FUNCTION_BLOCK ParallelUnits
VAR_INPUT
	EN: BOOL;
	Tags: REFERENCE TO AdsTagsParallelUnits;
	Parameters: REFERENCE TO GreenMasterBaseParameters;
END_VAR
VAR_OUTPUT
END_VAR
VAR
	LocalAmsNumber: LINT;
	RemoteAmsNumber: LINT;
	RemoteOrderToSend: RemoteOrder;
	RemoteStatusData: RemoteStatusData;
	Week: WORD;
	FirstTime: BOOL;
	HostName: FB_GetHostName;
	FoundHost: BOOL;
	StateTime: Timer;
	RemoteActive: BOOL;
	InstantaneousDualNeeded: BOOL;
	DualNeeded: BOOL;
	DualNeededTON: TON;
	DualNeededTOF: TOF;
	Runnable: BOOL;
	RemoteValidTOF: TOF;
	AddWeekTest: WORD;
	TransferOk: BOOL;
	TransferTON: TON;
	TempSP: LREAL;
	SupplyAirSetPointAdjustmentFB: SetPointAdjustmentFB;
	ExtractAirSetPointAdjustmentFB: SetPointAdjustmentFB;
	SupplyAirSetPointAdjustmentFB_HighSpeed: SetPointAdjustmentFB;
	ExtractAirSetPointAdjustmentFB_HighSpeed: SetPointAdjustmentFB;
	StandaloneSupplyAirSetPointAdjustmentFB: SetPointAdjustmentFB;
	StandaloneExtractAirSetPointAdjustmentFB: SetPointAdjustmentFB;
	StandaloneSupplyAirSetPointAdjustmentFB_HighSpeed: SetPointAdjustmentFB;
	StandaloneExtractAirSetPointAdjustmentFB_HighSpeed: SetPointAdjustmentFB;
END_VAR

IF NOT FirstTime THEN
	HostName(bExecute := TRUE);
	IF NOT HostName.bBusy THEN	
		FoundHost := FALSE;
		// E6
		IF F_ToUCase(HostName.sHostName) = 'STU_E6-LB01' THEN
			Tags.Settings.RemoteAmsId := '10.138.21.151.1.1';
			Tags.Status.isMaster := TRUE;
			FoundHost := TRUE;
		ELSIF F_ToUCase(HostName.sHostName) = 'STU_E6-LB02' THEN
			Tags.Settings.RemoteAmsId := '10.138.21.150.1.1';
			Tags.Status.isMaster := FALSE;
			FoundHost := TRUE;
		END_IF
		// E1
		IF F_ToUCase(HostName.sHostName) = 'STU_E1-LB01' THEN
			Tags.Settings.RemoteAmsId := '10.138.21.153.1.1';
			Tags.Status.isMaster := TRUE;
			FoundHost := TRUE;
		ELSIF F_ToUCase(HostName.sHostName) = 'STU_E1-LB02' THEN
			Tags.Settings.RemoteAmsId := '10.138.21.152.1.1';
			Tags.Status.isMaster := FALSE;
			FoundHost := TRUE;
		END_IF
		// DIGINET Test system
		IF F_ToUCase(HostName.sHostName) = 'DIGINET-1' THEN
			Tags.Settings.RemoteAmsId := '5.102.41.153.1.1';
			Tags.Status.isMaster := TRUE;
			FoundHost := TRUE;
		ELSIF F_ToUCase(HostName.sHostName) = 'DIGINET-2' THEN
			Tags.Settings.RemoteAmsId := '5.73.47.143.1.1';
			Tags.Status.isMaster := FALSE;
			FoundHost := TRUE;
		END_IF
		// NIBE AirSite Test system
		IF F_ToUCase(HostName.sHostName) = 'AIRPLC-DEMO' THEN
			Tags.Settings.RemoteAmsId := '5.102.42.161.1.1';
			Tags.Status.isMaster := TRUE;
			FoundHost := TRUE;
		ELSIF F_ToUCase(HostName.sHostName) = 'CX-662AA1' THEN
			Tags.Settings.RemoteAmsId := '10.133.0.22.1.1';
			Tags.Status.isMaster := FALSE;
			FoundHost := TRUE;
		END_IF
		IF NOT FoundHost THEN
			Tags.Status.isMaster := TRUE;			
		END_IF
		Tags.Status.isSlave := NOT Tags.Status.isMaster;
		// First time or remote AMS ID changed
		FirstTime := TRUE;
	END_IF
END_IF
StateTime();
Runnable := Parameters.System.Operation.State = SystemStates.Run;
IF Runnable THEN
	IF NOT InstantaneousDualNeeded THEN
		IF (Parameters.Regulation.SupplyAir.Control.CV > Tags.Settings.StandaloneMaxFan) OR
			(Parameters.Regulation.ExtractAir.Control.CV > Tags.Settings.StandaloneMaxFan) OR
			(RemoteStatusData.RemoteStatus.SupplyFanSpeed > Tags.Settings.StandaloneMaxFan) OR
			(RemoteStatusData.RemoteStatus.ExtractFanSpeed > Tags.Settings.StandaloneMaxFan) THEN
			InstantaneousDualNeeded := TRUE;
		END_IF
	ELSE
		IF (Parameters.Regulation.SupplyAir.Control.CV < Tags.Settings.DualMinFan) AND
			(Parameters.Regulation.ExtractAir.Control.CV < Tags.Settings.DualMinFan) AND
			(RemoteStatusData.RemoteStatus.SupplyFanSpeed < Tags.Settings.DualMinFan) AND
			(RemoteStatusData.RemoteStatus.ExtractFanSpeed < Tags.Settings.DualMinFan) THEN
			InstantaneousDualNeeded := FALSE;
		END_IF
	END_IF
	DualNeededTON(IN := InstantaneousDualNeeded, PT := T#5M);
	DualNeededTOF(IN := InstantaneousDualNeeded, PT := T#5M);
	IF NOT DualNeeded THEN
		IF DualNeededTON.Q THEN
			DualNeeded := TRUE;
		END_IF
	ELSE
		IF NOT DualNeededTOF.Q THEN
			DualNeeded := FALSE;
		END_IF
	END_IF
END_IF
Week := F_GetWeekOfTheYear(NowDT()) + AddWeekTest;;
RemoteValidTOF(IN := RemoteStatusData.Valid, PT := T#10S); 
RemoteActive := RemoteValidTOF.Q AND RemoteStatusData.RemoteStatus.IsRunning;
Tags.Status.SupplyFanSpeed := Parameters.Regulation.SupplyAir.Control.CV;
Tags.Status.ExtractFanSpeed := Parameters.Regulation.ExtractAir.Control.CV;
Tags.Status.IsRunning := Parameters.System.Operation.State = SystemStates.Run;
Tags.Status.ResetAlarm := Parameters.IO.DIn.ResetAlarm;
Tags.Status.Fire := Main.GreenMaster.FireAlarm();
Tags.Status.Freeze := Parameters.Alarm.Active.A.Freeze;
IF RemoteActive THEN
	Tags.Status.PressureSupplyCSP := GetSetPointSupply();
	Tags.Status.PressureExtractCSP := GetSetPointExtract();
ELSE
	Tags.Status.PressureSupplyCSP := GetStandaloneSetPointSupply();
	Tags.Status.PressureExtractCSP := GetStandaloneSetPointExtract();
END_IF

IF FirstTime THEN
	MasterSlave();
END_IF
IF EN THEN
	TransferTON(IN := TRUE, PT := T#1S);
	IF TransferTON.Q THEN
		TransferTON(IN := FALSE);
		RemoteStatusData := ReadFromRemote();
		IF RemoteStatusData.Valid THEN
			IF RemoteStatusData.RemoteStatus.ResetAlarm THEN
				Parameters.Alarm.Control.ResetAlarms := TRUE;
			END_IF
			RemoteOrderToSend.Counter := RemoteOrderToSend.Counter + 1;
			IF Tags.Status.IsMaster THEN
				RemoteOrderToSend.TimeChannels := Parameters.System.Operation.TimeChannels;
				RemoteOrderToSend.TemperatureControl := Parameters.Regulation.Temperature.Control;		
				RemoteOrderToSend.SupplyAirControl := Parameters.Regulation.SupplyAir.Control;		
				RemoteOrderToSend.ExtractAirControl := Parameters.Regulation.ExtractAir.Control;
				RemoteOrderToSend.TemperatureSetPointAdjustment := Parameters.Regulation.Temperature.SetPointAdjustment;
				RemoteOrderToSend.SupplyAirSetPointAdjustment := Parameters.Regulation.SupplyAir.SetPointAdjustment;
				RemoteOrderToSend.ExtractAirSetPointAdjustment := Parameters.Regulation.ExtractAir.SetPointAdjustment;
				RemoteOrderToSend.NightCoolingRequest := Parameters.Regulation.NightCoolingRequest;
			END_IF
			TransferOk := TransferToRemote(sNetId := Tags.Settings.RemoteAmsId, Src := RemoteOrderToSend, Dest := 'ADS_ParallelUnits.Tags.Settings.RemoteOrder');	
			IF TransferOk AND Tags.Status.IsSlave THEN
				Parameters.System.Operation.TimeChannels := Tags.Settings.RemoteOrder.TimeChannels;		
				Parameters.Regulation.Temperature.Control.SP := Tags.Settings.RemoteOrder.TemperatureControl.SP;		
				Parameters.Regulation.Temperature.Control.SP_HighSpeed := Tags.Settings.RemoteOrder.TemperatureControl.SP_HighSpeed;		
				Parameters.Regulation.SupplyAir.Control.SP := Tags.Settings.RemoteOrder.SupplyAirControl.SP;		
				Parameters.Regulation.SupplyAir.Control.SP_HighSpeed := Tags.Settings.RemoteOrder.SupplyAirControl.SP_HighSpeed;		
				Parameters.Regulation.ExtractAir.Control.SP := Tags.Settings.RemoteOrder.ExtractAirControl.SP;		
				Parameters.Regulation.ExtractAir.Control.SP_HighSpeed := Tags.Settings.RemoteOrder.ExtractAirControl.SP_HighSpeed;		
				Parameters.Regulation.Temperature.SetPointAdjustment := Tags.Settings.RemoteOrder.TemperatureSetPointAdjustment;		
				Parameters.Regulation.SupplyAir.SetPointAdjustment := Tags.Settings.RemoteOrder.SupplyAirSetPointAdjustment;		
				Parameters.Regulation.ExtractAir.SetPointAdjustment := Tags.Settings.RemoteOrder.ExtractAirSetPointAdjustment;	
				Parameters.Regulation.NightCoolingRequest := Tags.Settings.RemoteOrder.NightCoolingRequest;
			END_IF
		ELSE
			IF Tags.Status.IsSlave THEN
				Parameters.Regulation.NightCoolingRequest := FALSE;
			END_IF
		END_IF		
	END_IF
END_IF

METHOD GetAmsNumbers : BOOL
VAR_INPUT
END_VAR
VAR_INST
	LocalAddrBytes: AMSNETID;
	RemoteAddrBytes: AMSNETID;	
	FB_GetLocalAmsNetId: FB_GetLocalAmsNetId;
	UsedRemoteAmsId: string := '???';
END_VAR
IF Tags.Settings.RemoteAmsId <> UsedRemoteAmsId THEN
	UsedRemoteAmsId := Tags.Settings.RemoteAmsId;
	RemoteAddrBytes := F_ScanAmsNetIds(Tags.Settings.RemoteAmsId);
	FB_GetLocalAmsNetId(bExecute := TRUE, AddrBytes => LocalAddrBytes);
	FB_GetLocalAmsNetId(bExecute := FALSE);
	IF NOT FB_GetLocalAmsNetId.bBusy AND NOT FB_GetLocalAmsNetId.bError THEN			
		LocalAmsNumber := 	
						SHL(TO_LINT(LocalAddrBytes[0]),  40) + 
						SHL(TO_LINT(LocalAddrBytes[1]),  32) + 
						SHL(TO_LINT(LocalAddrBytes[2]),  24) + 
						SHL(TO_LINT(LocalAddrBytes[3]), 16) + 
						SHL(TO_LINT(LocalAddrBytes[4]), 8) + 
						TO_LINT(LocalAddrBytes[5]); 
		RemoteAmsNumber := 	
						SHL(TO_LINT(RemoteAddrBytes[0]),  40) + 
						SHL(TO_LINT(RemoteAddrBytes[1]),  32) + 
						SHL(TO_LINT(RemoteAddrBytes[2]),  24) + 
						SHL(TO_LINT(RemoteAddrBytes[3]), 16) + 
						SHL(TO_LINT(RemoteAddrBytes[4]), 8) + 
						TO_LINT(RemoteAddrBytes[5]); 
	END_IF
	GetAmsNumbers := TRUE;
ELSE 
	GetAmsNumbers := FALSE;
END_IF
END_METHOD

METHOD GetSetPointExtract : REAL
VAR_INPUT
END_VAR
VAR
	TempSP: REAL;
END_VAR
IF Parameters.Regulation.NightCooling OR Parameters.IO.DIn.ExtendedOperation OR Parameters.System.Operation.TimeChannels.HighSpeed THEN
	TempSP := Tags.Settings.PressureExtractSP_HighSpeed;
	ExtractAirSetPointAdjustmentFB_HighSpeed(X := Parameters.Regulation.CompensationTemperature, SetPointAdjustment := Tags.Settings.ExtractAirSetPointAdjustment_HighSpeed);
	GetSetPointExtract := TO_REAL(Tags.Settings.ExtractAirSetPointAdjustment_HighSpeed.Y) + TempSP;
ELSE
	TempSP := Tags.Settings.PressureExtractSP;
	ExtractAirSetPointAdjustmentFB(X := Parameters.Regulation.CompensationTemperature, SetPointAdjustment := Tags.Settings.ExtractAirSetPointAdjustment);
	GetSetPointExtract := TO_REAL(Tags.Settings.ExtractAirSetPointAdjustment.Y) + TempSP;
END_IF
END_METHOD

METHOD GetSetPointSupply : REAL
VAR_INPUT
END_VAR
VAR
	TempSP: REAL;
END_VAR
IF Parameters.Regulation.NightCooling OR Parameters.IO.DIn.ExtendedOperation OR Parameters.System.Operation.TimeChannels.HighSpeed THEN
	TempSP := Tags.Settings.PressureSupplySP_HighSpeed;
	SupplyAirSetPointAdjustmentFB_HighSpeed(X := Parameters.Regulation.CompensationTemperature, SetPointAdjustment := Tags.Settings.SupplyAirSetPointAdjustment_HighSpeed);
	GetSetPointSupply := TO_REAL(Tags.Settings.SupplyAirSetPointAdjustment_HighSpeed.Y) + TempSP;
ELSE
	TempSP := Tags.Settings.PressureSupplySP;
	SupplyAirSetPointAdjustmentFB(X := Parameters.Regulation.CompensationTemperature, SetPointAdjustment := Tags.Settings.SupplyAirSetPointAdjustment);
	GetSetPointSupply := TO_REAL(Tags.Settings.SupplyAirSetPointAdjustment.Y) + TempSP;
END_IF
END_METHOD

METHOD GetStandaloneSetPointExtract : REAL
VAR_INPUT
END_VAR
VAR
	TempSP: REAL;
END_VAR
IF Parameters.Regulation.NightCooling OR Parameters.IO.DIn.ExtendedOperation OR Parameters.System.Operation.TimeChannels.HighSpeed THEN
	TempSP := Tags.Settings.StandalonePressureExtractSP_HighSpeed;
	StandaloneExtractAirSetPointAdjustmentFB_HighSpeed(X := Parameters.Regulation.CompensationTemperature, SetPointAdjustment := Tags.Settings.StandaloneExtractAirSetPointAdjustment_HighSpeed);
	GetStandaloneSetPointExtract := TO_REAL(Tags.Settings.StandaloneExtractAirSetPointAdjustment_HighSpeed.Y) + TempSP;
ELSE
	TempSP := Tags.Settings.StandalonePressureExtractSP;
	StandaloneExtractAirSetPointAdjustmentFB(X := Parameters.Regulation.CompensationTemperature, SetPointAdjustment := Tags.Settings.StandaloneExtractAirSetPointAdjustment);
	GetStandaloneSetPointExtract := TO_REAL(Tags.Settings.StandaloneExtractAirSetPointAdjustment.Y) + TempSP;
END_IF
END_METHOD

METHOD GetStandaloneSetPointSupply : REAL
VAR_INPUT
END_VAR
VAR
	TempSP: REAL;
END_VAR
IF Parameters.Regulation.NightCooling OR Parameters.IO.DIn.ExtendedOperation OR Parameters.System.Operation.TimeChannels.HighSpeed THEN
	TempSP := Tags.Settings.StandalonePressureSupplySP_HighSpeed;
	StandaloneSupplyAirSetPointAdjustmentFB_HighSpeed(X := Parameters.Regulation.CompensationTemperature, SetPointAdjustment := Tags.Settings.StandaloneSupplyAirSetPointAdjustment_HighSpeed);
	GetStandaloneSetPointSupply := TO_REAL(Tags.Settings.StandaloneSupplyAirSetPointAdjustment_HighSpeed.Y) + TempSP;
ELSE
	TempSP := Tags.Settings.StandalonePressureSupplySP;
	StandaloneSupplyAirSetPointAdjustmentFB(X := Parameters.Regulation.CompensationTemperature, SetPointAdjustment := Tags.Settings.StandaloneSupplyAirSetPointAdjustment);
	GetStandaloneSetPointSupply := TO_REAL(Tags.Settings.StandaloneSupplyAirSetPointAdjustment.Y) + TempSP;
END_IF
END_METHOD

METHOD MasterSlave : BOOL
VAR_INPUT
END_VAR
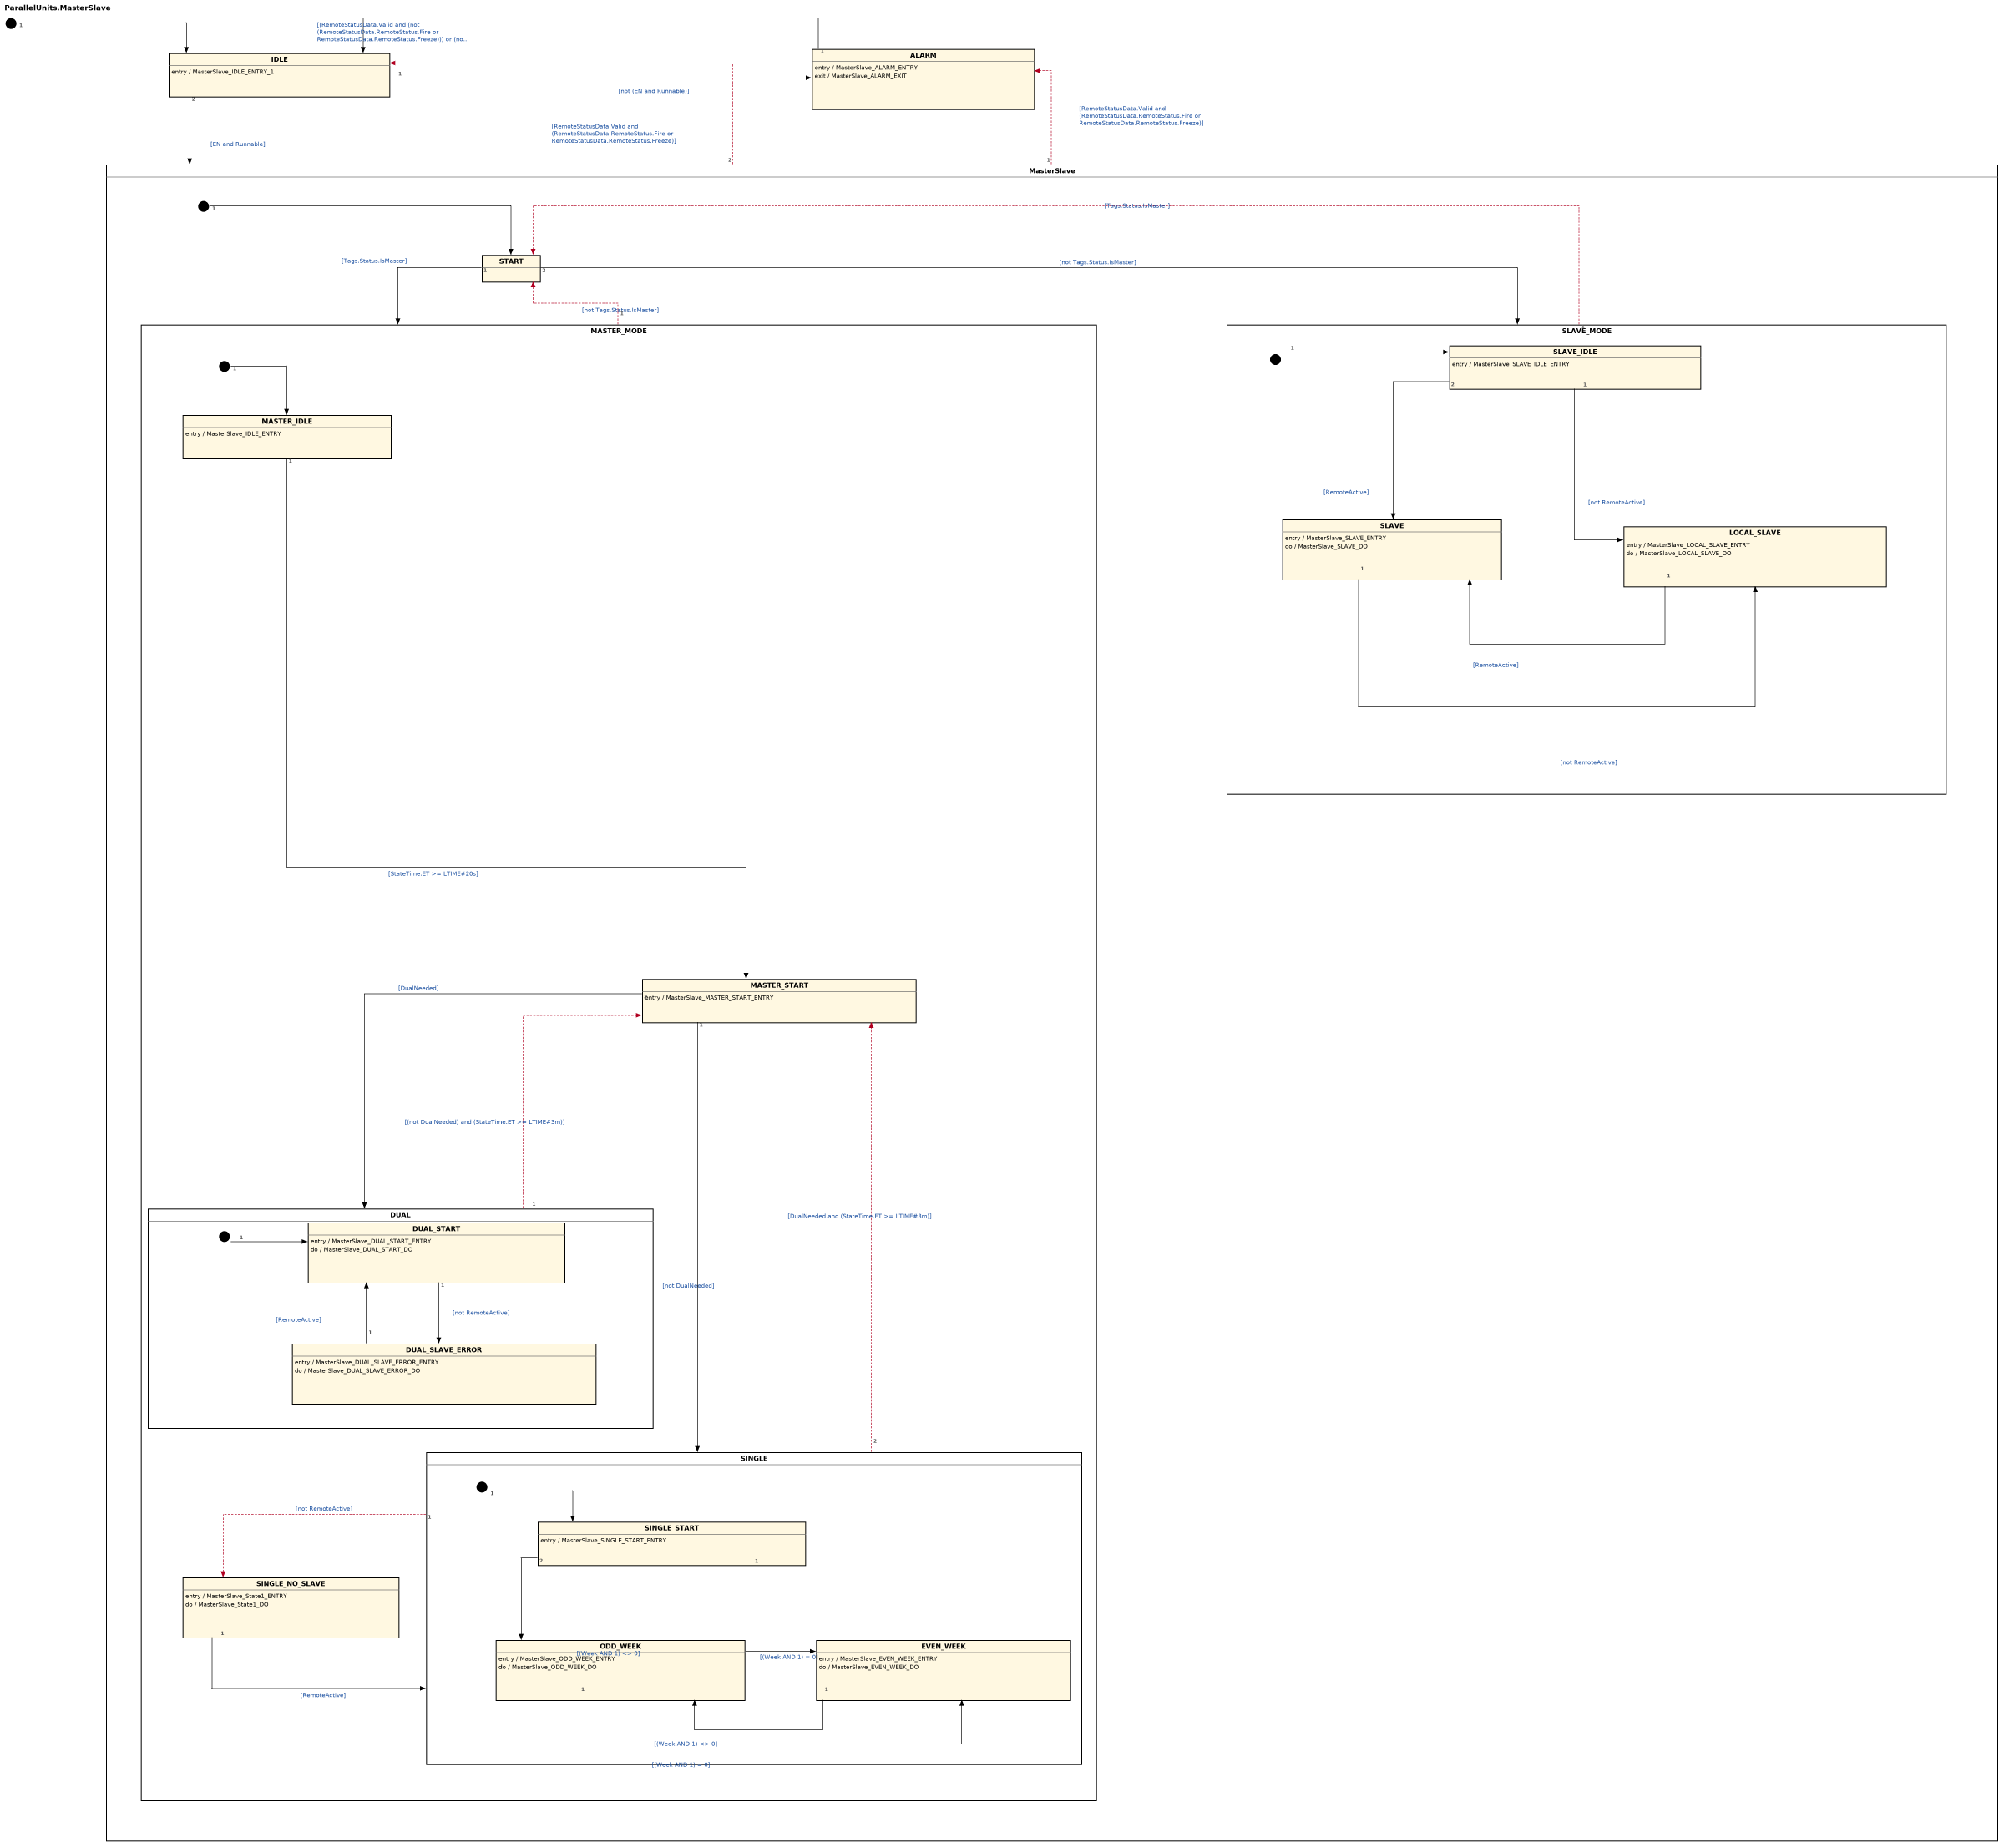
STATECHART MasterSlave  // abortable
    START StartState2
    STATE ALARM
        entry / MasterSlave_ALARM_ENTRY
        exit / MasterSlave_ALARM_EXIT
    STATE IDLE
        entry / MasterSlave_IDLE_ENTRY_1
    COMPOSITE STATE MasterSlave
        START StartState1
        STATE START
        COMPOSITE STATE MASTER_MODE
            START StartState6
            STATE MASTER_IDLE
                entry / MasterSlave_IDLE_ENTRY
            STATE MASTER_START
                entry / MasterSlave_MASTER_START_ENTRY
            COMPOSITE STATE DUAL
                START StartState4
                STATE DUAL_START
                    entry / MasterSlave_DUAL_START_ENTRY
                    do / MasterSlave_DUAL_START_DO
                STATE DUAL_SLAVE_ERROR
                    entry / MasterSlave_DUAL_SLAVE_ERROR_ENTRY
                    do / MasterSlave_DUAL_SLAVE_ERROR_DO
                StartState4 -> DUAL_START  // priority 1, on completion
                DUAL_START -> DUAL_SLAVE_ERROR [not RemoteActive] // priority 1
                DUAL_SLAVE_ERROR -> DUAL_START [RemoteActive] // priority 1
            END_STATE
            COMPOSITE STATE SINGLE
                START StartState3
                STATE SINGLE_START
                    entry / MasterSlave_SINGLE_START_ENTRY
                STATE ODD_WEEK
                    entry / MasterSlave_ODD_WEEK_ENTRY
                    do / MasterSlave_ODD_WEEK_DO
                STATE EVEN_WEEK
                    entry / MasterSlave_EVEN_WEEK_ENTRY
                    do / MasterSlave_EVEN_WEEK_DO
                StartState3 -> SINGLE_START  // priority 1, on completion
                SINGLE_START -> EVEN_WEEK [(Week AND 1) = 0] // priority 1
                SINGLE_START -> ODD_WEEK [(Week AND 1) <> 0] // priority 2
                ODD_WEEK -> EVEN_WEEK [(Week AND 1) = 0] // priority 1
                EVEN_WEEK -> ODD_WEEK [(Week AND 1) <> 0] // priority 1
            END_STATE
            STATE SINGLE_NO_SLAVE
                entry / MasterSlave_State1_ENTRY
                do / MasterSlave_State1_DO
            StartState6 -> MASTER_IDLE  // priority 1, on completion
            MASTER_IDLE -> MASTER_START [StateTime.ET >= LTIME#20s] // priority 1
            MASTER_START -> SINGLE [not DualNeeded] // priority 1
            MASTER_START -> DUAL [DualNeeded] // priority 2
            DUAL -> MASTER_START [(not DualNeeded) and (StateTime.ET >= LTIME#3m)] // priority 1, exception
            SINGLE -> SINGLE_NO_SLAVE [not RemoteActive] // priority 1, exception
            SINGLE -> MASTER_START [DualNeeded and (StateTime.ET >= LTIME#3m)] // priority 2, exception
            SINGLE_NO_SLAVE -> SINGLE [RemoteActive] // priority 1
        END_STATE
        COMPOSITE STATE SLAVE_MODE
            START StartState5
            STATE SLAVE_IDLE
                entry / MasterSlave_SLAVE_IDLE_ENTRY
            STATE SLAVE
                entry / MasterSlave_SLAVE_ENTRY
                do / MasterSlave_SLAVE_DO
            STATE LOCAL_SLAVE
                entry / MasterSlave_LOCAL_SLAVE_ENTRY
                do / MasterSlave_LOCAL_SLAVE_DO
            StartState5 -> SLAVE_IDLE  // priority 1, on completion
            SLAVE_IDLE -> LOCAL_SLAVE [not RemoteActive] // priority 1
            SLAVE_IDLE -> SLAVE [RemoteActive] // priority 2
            SLAVE -> LOCAL_SLAVE [not RemoteActive] // priority 1
            LOCAL_SLAVE -> SLAVE [RemoteActive] // priority 1
        END_STATE
        StartState1 -> START  // priority 1, on completion
        START -> MASTER_MODE [Tags.Status.IsMaster] // priority 1
        START -> SLAVE_MODE [not Tags.Status.IsMaster] // priority 2
        MASTER_MODE -> START [not Tags.Status.IsMaster] // priority 1, exception
        SLAVE_MODE -> START [Tags.Status.IsMaster] // priority 1, exception
    END_STATE
    StartState2 -> IDLE  // priority 1, on completion
    ALARM -> IDLE [(RemoteStatusData.Valid and (not (RemoteStatusData.RemoteStatus.Fire or RemoteStatusData.RemoteStatus.Freeze))) or (not RemoteStatusData.Valid)] // priority 1
    IDLE -> ALARM [RemoteStatusData.Valid and (RemoteStatusData.RemoteStatus.Fire or RemoteStatusData.RemoteStatus.Freeze)] // priority 1
    IDLE -> MasterSlave [EN and Runnable] // priority 2
    MasterSlave -> ALARM [RemoteStatusData.Valid and (RemoteStatusData.RemoteStatus.Fire or RemoteStatusData.RemoteStatus.Freeze)] // priority 1, exception
    MasterSlave -> IDLE [not (EN and Runnable)] // priority 2, exception
END_STATECHART
END_METHOD

METHOD MasterSlave_ALARM_ENTRY : BOOL
VAR_INPUT
END_VAR
Parameters.System.Operation.EN := FALSE;
END_METHOD

METHOD MasterSlave_ALARM_EXIT : BOOL
VAR_INPUT
END_VAR
Parameters.System.Operation.EN := TRUE;
END_METHOD

METHOD MasterSlave_DUAL_SLAVE_ERROR_DO : BOOL
VAR_INPUT
END_VAR
Parameters.Regulation.SupplyAir.Control.SP := GetStandaloneSetPointSupply();
Parameters.Regulation.ExtractAir.Control.SP := GetStandaloneSetPointExtract();
END_METHOD

METHOD MasterSlave_DUAL_SLAVE_ERROR_ENTRY : BOOL
VAR_INPUT
END_VAR
Parameters.Regulation.SupplyAir.ControlMode := FanControlTypes.Pressure;
Parameters.Regulation.ExtractAir.ControlMode := FanControlTypes.Pressure;
END_METHOD

METHOD MasterSlave_DUAL_START_DO : BOOL
VAR_INPUT
END_VAR
Parameters.Regulation.SupplyAir.Control.SP := PidControlSupplyAir(Sync := FALSE, SyncCV := 0);
Parameters.Regulation.ExtractAir.Control.SP := PidControlExtractAir(Sync := FALSE, SyncCV := 0);
RemoteOrderToSend.SupplySP := Parameters.Regulation.SupplyAir.Control.SP;
RemoteOrderToSend.ExtractSP := Parameters.Regulation.ExtractAir.Control.SP;
END_METHOD

METHOD MasterSlave_DUAL_START_ENTRY : BOOL
VAR_INPUT
END_VAR
StateTime.Restart();
Parameters.IO.DOut.T_QM2 := TRUE;
Parameters.IO.DOut.F_QM1 := TRUE;	
Parameters.Regulation.SupplyAir.ControlMode := FanControlTypes.Const;
Parameters.Regulation.ExtractAir.ControlMode := FanControlTypes.Const;
PidControlSupplyAir(Sync := FALSE, SyncCV := 0.55);
PidControlExtractAir(Sync := FALSE, SyncCV := 0.65);
PidControlSupplyAir(Sync := TRUE, SyncCV := 0.55);
PidControlExtractAir(Sync := TRUE, SyncCV := 0.65);
END_METHOD

METHOD MasterSlave_EVEN_WEEK_DO : BOOL
VAR_INPUT
END_VAR
Parameters.Regulation.SupplyAir.Control.SP := 0;
Parameters.Regulation.ExtractAir.Control.SP := 0;
RemoteOrderToSend.SupplySP := PidControlSupplyAir(Sync := FALSE, SyncCV := 0);
RemoteOrderToSend.ExtractSP := PidControlExtractAir(Sync := FALSE, SyncCV := 0);
END_METHOD

METHOD MasterSlave_EVEN_WEEK_ENTRY : BOOL
VAR_INPUT
END_VAR
Parameters.IO.DOut.T_QM2 := FALSE;
Parameters.IO.DOut.F_QM1 := FALSE;
END_METHOD

ACTION MasterSlave_IDLE_ENTRY:
StateTime.Restart();
Tags.Status.MasterActive := TRUE;
END_ACTION

METHOD MasterSlave_IDLE_ENTRY_1 : BOOL
VAR_INPUT
END_VAR
Parameters.Regulation.SupplyAir.ControlMode := FanControlTypes.Const;
Parameters.Regulation.ExtractAir.ControlMode := FanControlTypes.Const;
Parameters.Regulation.SupplyAir.Control.SP := 0;
Parameters.Regulation.ExtractAir.Control.SP := 0;
Tags.Settings.RemoteOrder.SupplySP := 0;
Tags.Settings.RemoteOrder.ExtractSP := 0;
END_METHOD

METHOD MasterSlave_LOCAL_ENTRY : BOOL
VAR_INPUT
END_VAR
Parameters.System.Operation.EN := TRUE;
Parameters.Regulation.SupplyAir.ControlMode := FanControlTypes.Pressure;
Parameters.Regulation.ExtractAir.ControlMode := FanControlTypes.Pressure;
Parameters.Regulation.SupplyAir.Control.SP := GetStandaloneSetPointSupply();
Parameters.Regulation.ExtractAir.Control.SP := GetStandaloneSetPointExtract();
END_METHOD

METHOD MasterSlave_LOCAL_SLAVE_DO : BOOL
VAR_INPUT
END_VAR
Parameters.Regulation.SupplyAir.Control.SP := GetStandaloneSetPointSupply();
Parameters.Regulation.ExtractAir.Control.SP := GetStandaloneSetPointExtract();
END_METHOD

METHOD MasterSlave_LOCAL_SLAVE_ENTRY : BOOL
VAR_INPUT
END_VAR
Parameters.Regulation.SupplyAir.ControlMode := FanControlTypes.Pressure;
Parameters.Regulation.ExtractAir.ControlMode := FanControlTypes.Pressure;
Parameters.IO.DOut.T_QM2 := TRUE;
Parameters.IO.DOut.F_QM1 := TRUE;
END_METHOD

METHOD MasterSlave_MANUAL_ENTRY : BOOL
VAR_INPUT
END_VAR
Parameters.Regulation.SupplyAir.ControlMode := FanControlTypes.Pressure;
Parameters.Regulation.ExtractAir.ControlMode := FanControlTypes.Pressure;
Parameters.Regulation.SupplyAir.Control.SP := GetSetPointSupply();
Parameters.Regulation.ExtractAir.Control.SP := GetSetPointExtract();
END_METHOD

METHOD MasterSlave_MASTER_START_ENTRY : BOOL
VAR_INPUT
END_VAR
StateTime.Restart();
PidControlSupplyAir(Sync := FALSE, SyncCV := 0);
PidControlExtractAir(Sync := false, SyncCV := 0);
PidControlSupplyAir(Sync := TRUE, SyncCV := 0);
PidControlExtractAir(Sync := TRUE, SyncCV := 0);
END_METHOD

METHOD MasterSlave_ODD_WEEK_DO : BOOL
VAR_INPUT
END_VAR
Parameters.Regulation.SupplyAir.Control.SP := PidControlSupplyAir(Sync := FALSE, SyncCV := 0);
Parameters.Regulation.ExtractAir.Control.SP := PidControlExtractAir(Sync := FALSE, SyncCV := 0);
RemoteOrderToSend.SupplySP := 0;
RemoteOrderToSend.ExtractSP := 0;
END_METHOD

METHOD MasterSlave_ODD_WEEK_ENTRY : BOOL
VAR_INPUT
END_VAR
Parameters.IO.DOut.T_QM2 := TRUE;
Parameters.IO.DOut.F_QM1 := TRUE;
END_METHOD

METHOD MasterSlave_SINGLE_START_ENTRY : BOOL
VAR_INPUT
END_VAR
StateTime.Restart();
Parameters.Regulation.SupplyAir.ControlMode := FanControlTypes.Const;
Parameters.Regulation.ExtractAir.ControlMode := FanControlTypes.Const;
PidControlSupplyAir(Sync := FALSE, SyncCV := 0.55);
PidControlExtractAir(Sync := false, SyncCV := 0.65);
PidControlSupplyAir(Sync := TRUE, SyncCV := 0.55);
PidControlExtractAir(Sync := TRUE, SyncCV := 0.65);
END_METHOD

METHOD MasterSlave_SLAVE_DO : BOOL
VAR_INPUT
END_VAR
VAR
	Supply: LREAL;
	Extract: LREAL;
END_VAR
Parameters.Regulation.SupplyAir.Control.SP := Tags.Settings.RemoteOrder.SupplySP;
Parameters.Regulation.ExtractAir.Control.SP := Tags.Settings.RemoteOrder.ExtractSP;	
IF (Tags.Settings.RemoteOrder.SupplySP = 0) AND (Tags.Settings.RemoteOrder.ExtractSP = 0) THEN
	Parameters.IO.DOut.T_QM2 := FALSE;
	Parameters.IO.DOut.F_QM1 := FALSE;	
ELSE
	Parameters.IO.DOut.T_QM2 := TRUE;
	Parameters.IO.DOut.F_QM1 := TRUE;	
END_IF
END_METHOD

METHOD MasterSlave_SLAVE_ENTRY : BOOL
VAR_INPUT
END_VAR
StateTime.Restart();
Parameters.Regulation.SupplyAir.ControlMode := FanControlTypes.Const;
Parameters.Regulation.ExtractAir.ControlMode := FanControlTypes.Const;
END_METHOD

METHOD MasterSlave_SLAVE_IDLE_ENTRY : BOOL
VAR_INPUT
END_VAR
StateTime.Restart();
END_METHOD

METHOD MasterSlave_State1_DO : BOOL
VAR_INPUT
END_VAR
Parameters.Regulation.SupplyAir.Control.SP := GetStandaloneSetPointSupply();
Parameters.Regulation.ExtractAir.Control.SP := GetStandaloneSetPointExtract();
END_METHOD

METHOD MasterSlave_State1_ENTRY : BOOL
VAR_INPUT
END_VAR
Parameters.Regulation.SupplyAir.ControlMode := FanControlTypes.Pressure;
Parameters.Regulation.ExtractAir.ControlMode := FanControlTypes.Pressure;
Parameters.IO.DOut.T_QM2 := TRUE;
Parameters.IO.DOut.F_QM1 := TRUE;
END_METHOD

METHOD PidControlExtractAir : LREAL
VAR_INPUT
	Sync: BOOL;
	SyncCV: LREAL := 0;
END_VAR
VAR_INST
	pid: PidController;
	pidOutput: LREAL;
END_VAR
pid(	SP := GetSetPointExtract(), 
		PV := Parameters.IO.AIn.F_BP1, 
		Sync := Sync, 
		SyncCV := SyncCV,
		P := Tags.Settings.Kp, 
		I := Tags.Settings.fTn, 
		DampingTime := Tags.Settings.fTv, 
		CV => pidOutput);
PidControlExtractAir := LimitValue(pidOutput * 100, 0, 100);
END_METHOD

METHOD PidControlSupplyAir : LREAL
VAR_INPUT
	Sync: BOOL;
	SyncCV: LREAL := 0;
END_VAR
VAR_INST
	pid: PidController;
	pidOutput: LREAL;
END_VAR
pid(	SP := GetSetPointSupply(), 
		PV := Parameters.IO.AIn.T_BP1, 
		Sync := Sync, 
		SyncCV := SyncCV,
		P := Tags.Settings.Kp, 
		I := Tags.Settings.fTn, 
		DampingTime := Tags.Settings.fTv, 
		CV => pidOutput);
PidControlSupplyAir := LimitValue(pidOutput * 100, 0, 100);
END_METHOD

METHOD ReadFromRemote : RemoteStatusData
VAR_INPUT
END_VAR
VAR_INST
	ReadAdsSymbol:FB_ReadAdsSymByName;	
	RemoteStatus: ParallelUnitsStatus;
	ValidTOF: TOF;
END_VAR
IF NOT ReadAdsSymbol.bBusy THEN
	ReadAdsSymbol(	bRead		:=	TRUE,
					sNetId		:=	Tags.Settings.RemoteAmsId,
					nPort		:=	851,
					sVarName	:=	'ADS_ParallelUnits.Tags.Status',
					nDestAddr	:=	ADR(RemoteStatus),
					nLen		:=	SIZEOF(RemoteStatus),
					tTimeout	:=	DEFAULT_ADS_TIMEOUT,
					eComMode	:=	eAdsComModeFastCom);
END_IF;
ReadAdsSymbol(bRead := FALSE);
ValidTOF(IN := NOT ReadAdsSymbol.bBusy AND NOT ReadAdsSymbol.bError, PT := T#5S);
ReadFromRemote.Valid := ValidTOF.Q;
ReadFromRemote.RemoteStatus := RemoteStatus;
END_METHOD

METHOD TransferToRemote : BOOL
VAR_INPUT
	sNetId: T_AmsNetID;
	Src: REFERENCE TO RemoteOrder;
	Dest: string;
END_VAR
VAR_INST
	WriteAdsSymbol: FB_WriteAdsSymByName;	
END_VAR
IF NOT WriteAdsSymbol.bBusy THEN
	WriteAdsSymbol(	bWrite		:=	TRUE,
					sNetId		:=	Tags.Settings.RemoteAmsId,
					nPort		:=	851,
					sVarName	:=	Dest,
					nSrcAddr	:=	ADR(Src),
					nLen		:=	SIZEOF(Src),
					tTimeout	:=	DEFAULT_ADS_TIMEOUT,
					eComMode	:=	eAdsComModeFastCom);
END_IF;
WriteAdsSymbol(bWrite := FALSE);
TransferToRemote := NOT WriteAdsSymbol.bBusy AND NOT WriteAdsSymbol.bError;
END_METHOD

END_FUNCTION_BLOCK

(* stored: Version 1.1.0.1, ProductVersion 3.1.4024.6
   POU ParallelUnits: Id {2de2df00-dc30-47a3-820e-7a0728f9500d}, SpecialFunc None
   Method GetAmsNumbers: Id {8b184dae-b98f-437b-b887-218bcb47a5ae}
   Method GetSetPointExtract: Id {c29c6065-5247-430e-b72e-7ac9718a871e}
   Method GetSetPointSupply: Id {c3ee25e9-905b-418f-8441-5da5cfd2f92b}
   Method GetStandaloneSetPointExtract: Id {b420f3aa-2fc5-4322-8fed-de5f672d61f0}
   Method GetStandaloneSetPointSupply: Id {1f6f6f04-f101-4d85-9dc1-bd41648f4a2f}
   Method MasterSlave: Id {b067a2be-016b-43dd-9bed-2081b3598c68}
   Method MasterSlave_ALARM_ENTRY: Id {2ef1aabf-ebaa-42ef-aeaf-b225c6846741}
   Method MasterSlave_ALARM_EXIT: Id {6e2443c7-f7c7-48f2-8ae1-7eb9b54f0df0}
   Method MasterSlave_DUAL_SLAVE_ERROR_DO: Id {ffea7271-2cec-4f36-8b1e-f1653e1f95fd}
   Method MasterSlave_DUAL_SLAVE_ERROR_ENTRY: Id {a41c604e-7dfe-46c1-92c3-320c97241782}
   Method MasterSlave_DUAL_START_DO: Id {ef1085be-0a80-4af2-9939-ff693c539123}
   Method MasterSlave_DUAL_START_ENTRY: Id {8b2ffe7d-9039-4405-bc94-9d525f03229b}
   Method MasterSlave_EVEN_WEEK_DO: Id {cd5dec14-245f-4c3d-9715-9c9ef56cc3bb}
   Method MasterSlave_EVEN_WEEK_ENTRY: Id {cdfb2ff3-6efc-4241-ac51-209da2003b94}
   Action MasterSlave_IDLE_ENTRY: Id {0312e5d5-7d85-4238-8c5e-05d62177278d}
   Method MasterSlave_IDLE_ENTRY_1: Id {f352ac4e-2cfc-451a-897b-693465e515d8}
   Method MasterSlave_LOCAL_ENTRY: Id {a17161f3-8041-4a38-a74a-14abd7306eb4}
   Method MasterSlave_LOCAL_SLAVE_DO: Id {60f718a8-c7ab-49e8-9a18-69d33378bab8}
   Method MasterSlave_LOCAL_SLAVE_ENTRY: Id {18e41049-1678-4fe4-b251-aace6ad405f9}
   Method MasterSlave_MANUAL_ENTRY: Id {6e8420de-9bd4-4de8-853c-e5fdc885b9c0}
   Method MasterSlave_MASTER_START_ENTRY: Id {13105fd1-a1eb-4695-ba2f-55e83b39354b}
   Method MasterSlave_ODD_WEEK_DO: Id {6fbd1167-84b7-4aae-bc41-61d7dad8a81a}
   Method MasterSlave_ODD_WEEK_ENTRY: Id {4a3a8e13-05d0-4e11-a6e4-905a71a2a288}
   Method MasterSlave_SINGLE_START_ENTRY: Id {cfb59907-89bf-4cf6-8927-54290e569e82}
   Method MasterSlave_SLAVE_DO: Id {6f870cc6-f864-4a4f-b92e-73aa64aa9f8d}
   Method MasterSlave_SLAVE_ENTRY: Id {57dfdd2f-5936-4441-ad52-666e43930558}
   Method MasterSlave_SLAVE_IDLE_ENTRY: Id {4d5f68dd-6ca9-4558-9f07-03c2bfb8d16d}
   Method MasterSlave_State1_DO: Id {6f1c77c3-572d-40d8-b63c-d2b8be28c94d}
   Method MasterSlave_State1_ENTRY: Id {3d9415ce-7612-4dd8-ad74-51df65abbfab}
   Method PidControlExtractAir: Id {c8594678-9bf4-440c-8f52-063a516084c6}
   Method PidControlSupplyAir: Id {190391ff-3d8b-4f81-bcde-0da9556bd2b7}
   Method ReadFromRemote: Id {c6962458-7669-4f7b-8fb6-3c1284286952}
   Method TransferToRemote: Id {60cfede9-10bb-4159-93d4-39b9dec23d1c} *)
